// Mitsubishi GX Works2 project: 240507_timechart11_한번on두번off3   PLC: Q03UDV

PROGRAM MAIN
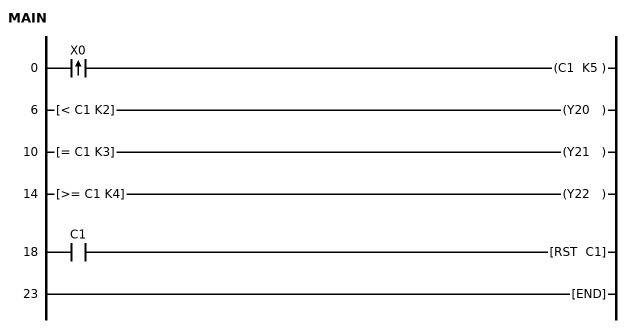
0     LDP     X0
      OUT     C1 K5
6     LD<     C1 K2
      OUT     Y20
10    LD=     C1 K3
      OUT     Y21
14    LD>=    C1 K4
      OUT     Y22
18    LD      C1
      RST     C1
23    END
END_PROGRAM
